FUNCTION_BLOCK FB_HeatpumpInit
VAR_IN_OUT
	MBMaster		:	ModbusRtuMasterV2_KL6x22B;
	Get				:	ST_HeatpumpGet;
END_VAR

VAR_INPUT
	ACPowerStatus	:	BOOL;
	HeatPumpID		:	BYTE;
	SFCInit			:	BOOL;
END_VAR
		
VAR
	TransmissionDone		:	BOOL;
	DataBuffer				:	ARRAY[0..50] OF WORD;
	b_MBBusy				:	BOOL;
	b_MBerr					:	BOOL;
	ui_cbRead				:	UINT;
	b_EnableTransmission	:	BOOL;
	ModbusRetryTimer		:	TON := (PT := TIME#250MS);
	ModbusStartTrigger		:	R_Trig;
	TransmissionDoneTrigger	:	F_Trig;
	MBRetryCount			:	BYTE;
	u_Counter				:	uint;
	
	SendValue		:	WORD;
	
	w_errid: Tc2_ModbusRTU.MODBUS_ERRORS;
	ResetRetryTimer: BOOL;
END_VAR
VAR_OUTPUT
END_VAR
VAR
END_VAR

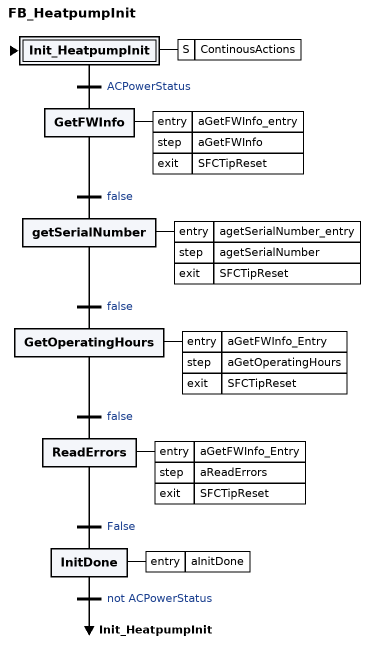
INITIAL_STEP Init_HeatpumpInit:
    ContinousActions(S);
END_STEP
TRANSITION FROM Init_HeatpumpInit TO GetFWInfo
    := ACPowerStatus;
END_TRANSITION
STEP GetFWInfo:
    aGetFWInfo_entry(P1);  // entry action
    aGetFWInfo(N);  // step action
    SFCTipReset(P0);  // exit action
END_STEP
TRANSITION FROM GetFWInfo TO getSerialNumber
    := false;
END_TRANSITION
STEP getSerialNumber:
    agetSerialNumber_entry(P1);  // entry action
    agetSerialNumber(N);  // step action
    SFCTipReset(P0);  // exit action
END_STEP
TRANSITION FROM getSerialNumber TO GetOperatingHours
    := false;
END_TRANSITION
STEP GetOperatingHours:
    aGetFWInfo_Entry(P1);  // entry action
    aGetOperatingHours(N);  // step action
    SFCTipReset(P0);  // exit action
END_STEP
TRANSITION FROM GetOperatingHours TO ReadErrors
    := false;
END_TRANSITION
STEP ReadErrors:
    aGetFWInfo_Entry(P1);  // entry action
    aReadErrors(N);  // step action
    SFCTipReset(P0);  // exit action
END_STEP
TRANSITION FROM ReadErrors TO InitDone
    := False;
END_TRANSITION
STEP InitDone:
    aInitDone(P1);  // entry action
END_STEP
TRANSITION FROM InitDone TO Init_HeatpumpInit
    := not ACPowerStatus;
END_TRANSITION

ACTION aGetFWInfo:

//ModbusStartTrigger(clk := b_EnableTransmission);

IF NOT b_enableTransmission THEN
	b_enableTransmission := TRUE;
END_IF

MBMaster.ReadRegs(	UnitID 		:= 	HeatPumpID,
					Quantity 	:= 	4,
					MBAddr		:=	1,
					cbLength 	:= 	64,
					pMemoryAddr	:=	ADR(DataBuffer),
					Execute		:=	ModbusStartTrigger.Q,
					Timeout		:=	T#250MS,		
					Busy		=>	b_MBBusy,
					Error 		=>	b_MBerr,
					cbRead 		=>	ui_cbRead,
					ErrorId		=>	w_errid
					);


TransmissionDoneTrigger(clk := b_MBBusy);

IF TransmissionDoneTrigger.q THEN
	IF NOT b_MBerr THEN
		get.HeatpumpData.i_FW_Version 		:= 	WORD_TO_INT(DataBuffer[0]);
		get.HeatpumpData.i_FW_release 		:= 	WORD_TO_INT(DataBuffer[1]);
		get.HeatpumpData.w_FW_Subrelease 	:= 	DataBuffer[2];
		get.HeatpumpData.w_FW_creationDate	:=	DataBuffer[3];
			
		TransmissionDone := TRUE;
		//done, preset for next step
		//b_EnableTransmission := FALSE;
		//ModbusStartTrigger(clk := b_EnableTransmission);
		MBRetryCount := 0;
		//ResetRetryTimer := TRUE;
		
		sfctip := TRUE;
	ELSE
		MBRetryCount := MBRetryCount + 1;
		b_EnableTransmission	:= FALSE;
		
		//if heatpump is still unreachable after 1 minute, something failed during poweron
		IF MBRetryCount > 240 THEN
			get.HeatPumpState := eHeatpumpState.ERROR;
			get.Events.b_CommError := TRUE;
		END_IF
	END_IF
END_IF



(*
IF b_EnableTransmission AND NOT b_MBBusy[0] THEN
	IF NOT b_MBerr[0] THEN
			//transmission done, process data
			get.HeatpumpData.i_FW_Version 		:= 	WORD_TO_INT(DataBuffer[0]);
			get.HeatpumpData.i_FW_release 		:= 	WORD_TO_INT(DataBuffer[1]);
			get.HeatpumpData.w_FW_Subrelease 	:= 	DataBuffer[2];
			get.HeatpumpData.w_FW_creationDate	:=	DataBuffer[3];
			
			TransmissionDone := TRUE;
			//done, preset for next step
			//b_EnableTransmission := FALSE;
			//ModbusStartTrigger(clk := b_EnableTransmission);
			MBRetryCount := 0;
	
			//sfctip := TRUE;
		ELSE
			MBRetryCount := MBRetryCount + 1;
			
			//add comm error functionality later
			IF MBRetryCount < 10 THEN
				//retry
				b_EnableTransmission	:= FALSE;
			ELSE
				//do something else
				b_EnableTransmission	:= FALSE;
			END_IF
		END_IF
	END_IF


IF TransmissionDone THEN
	sfctip := TRUE;
END_IF


IF NOT b_MBBusy[0] THEN
	IF NOT b_MBerr[0] THEN
		//transmission done, process data
		get.HeatpumpData.i_FW_Version 		:= 	WORD_TO_INT(DataBuffer[0]);
		get.HeatpumpData.i_FW_release 		:= 	WORD_TO_INT(DataBuffer[1]);
		get.HeatpumpData.w_FW_Subrelease 	:= 	DataBuffer[2];
		get.HeatpumpData.w_FW_creationDate	:=	DataBuffer[3];
		
		//done, preset for next step
		b_EnableTransmission := FALSE;
		ModbusStartTrigger(clk := b_EnableTransmission);
		MBRetryCount := 0;

		sfctip := TRUE;
	ELSE
		MBRetryCount := MBRetryCount + 1;
		
		//add comm error functionality later
		IF MBRetryCount < 10 THEN
			//retry
			b_EnableTransmission	:= FALSE;
		ELSE
			//do something else
			b_EnableTransmission	:= FALSE;
		END_IF
	END_IF
END_IF
*)
END_ACTION

ACTION aGetFWInfo_entry:
//ResetRetryTimer := TRUE;
//TransmissionDone := False;

get.HeatPumpState := eHeatpumpState.Initializing;
END_ACTION

ACTION aGetOperatingHours:


MBMaster.ReadRegs(	UnitID 		:= 	HeatPumpID,
					Quantity 	:= 	1,
					MBAddr		:=	305,
					cbLength 	:= 	1*2,
					pMemoryAddr	:=	ADR(DataBuffer),
					Execute		:=	ModbusStartTrigger.Q,
					Timeout		:=	T#250MS,		
					Busy		=>	b_MBBusy,
					Error 		=>	b_MBerr,
					cbRead 		=>	ui_cbRead,
					ErrorId		=>	w_errid
					);

TransmissionDoneTrigger(clk := b_MBBusy);

IF TransmissionDoneTrigger.q THEN
	IF NOT b_MBerr THEN
		//transmission done, process data
		
		//just use comp 1 for now. See if the others are even used
		//i think it will be a dual word value. But check later
		get.HeatpumpData.i_OperatingHours := WORD_TO_INT(DataBuffer[0]);
		
		//done, preset for next step
		b_EnableTransmission := FALSE;
//		ModbusStartTrigger(clk := b_EnableTransmission);
		MBRetryCount := 0;
		sfctip := TRUE;
	ELSE
		MBRetryCount := MBRetryCount + 1;
		b_EnableTransmission	:= FALSE;
		
		//if comm fails 5 times in a row. system is unusable
		IF MBRetryCount > 5 THEN
			get.HeatPumpState := eHeatpumpState.ERROR;
			get.Events.b_CommError := TRUE;
		END_IF
	END_IF
END_IF
END_ACTION

ACTION agetSerialNumber:



IF NOT b_enableTransmission THEN
	b_enableTransmission := TRUE;
END_IF


MBMaster.ReadRegs(	UnitID 		:= 	HeatPumpID,
					Quantity 	:= 	18,
					MBAddr		:=	80,
					cbLength 	:= 	32*2,
					pMemoryAddr	:=	ADR(DataBuffer),
					Execute		:=	ModbusStartTrigger.Q,
					Timeout		:=	T#250MS,		
					Busy		=>	b_MBBusy,
					Error 		=>	b_MBerr,
					cbRead 		=>	ui_cbRead,
					ErrorId		=>	w_errid
					);

TransmissionDoneTrigger(clk := b_MBBusy);

IF TransmissionDoneTrigger.q THEN
	IF NOT b_MBerr THEN
		FOR u_counter:=0 TO 17 BY 1 DO
			get.HeatpumpData.w_Serialnumber[u_counter]	:= 	DataBuffer[u_counter];
		END_FOR
			
		TransmissionDone := TRUE;
		//done, preset for next step
		//b_EnableTransmission := FALSE;
		//ModbusStartTrigger(clk := b_EnableTransmission);
		MBRetryCount := 0;
	
		sfctip := TRUE;
	ELSE
		MBRetryCount := MBRetryCount + 1;
		b_EnableTransmission	:= FALSE;
		
		//if comm fails 5 times in a row. system is unusable
		IF MBRetryCount > 5 THEN
			get.HeatPumpState := eHeatpumpState.ERROR;
			get.Events.b_CommError := TRUE;
		END_IF
	END_IF
END_IF

(*
IF b_EnableTransmission AND NOT b_MBBusy[2] THEN
	IF NOT b_MBerr[2] THEN
		//transmission done, process data

		
		//maybe try to put get struct directly in MBREAD pMemoryAddr later
		FOR u_counter:=0 TO 8 BY 1 DO
			get.HeatpumpData.w_Serialnumber[u_counter]	:= 	DataBuffer[u_counter];
		END_FOR
			
			TransmissionDone := TRUE;
			//done, preset for next step
			//b_EnableTransmission := FALSE;
			//ModbusStartTrigger(clk := b_EnableTransmission);
			MBRetryCount := 0;
	
			//sfctip := TRUE;
		ELSE
			MBRetryCount := MBRetryCount + 1;
			
			//add comm error functionality later
			IF MBRetryCount < 10 THEN
				//retry
				b_EnableTransmission	:= FALSE;
			ELSE
				//do something else
				b_EnableTransmission	:= FALSE;
			END_IF
		END_IF
	END_IF


IF TransmissionDone THEN
	sfctip := TRUE;
END_IF
		
				
IF NOT b_MBBusy[2] THEN
	IF NOT b_MBerr[2] THEN
		//transmission done, process data
		
		//maybe try to put get struct directly in MBREAD pMemoryAddr later
		FOR u_counter:=0 TO 8 BY 1 DO
			get.HeatpumpData.w_Serialnumber[u_counter]	:= 	DataBuffer[u_counter];
		END_FOR
		
		//done, preset for next step
		b_EnableTransmission := FALSE;
		ModbusStartTrigger(clk := b_EnableTransmission);
		MBRetryCount := 0;
		sfctip := TRUE;
	ELSE
		MBRetryCount := MBRetryCount + 1;
		
		//add comm error functionality later
		IF MBRetryCount < 10 THEN
			//retry
			b_EnableTransmission	:= FALSE;
		ELSE
			//do something else
			b_EnableTransmission	:= FALSE;
		END_IF
	END_IF
END_IF
*)
END_ACTION

ACTION agetSerialNumber_entry:
//SFCTip := FALSE;
//TransmissionDone := False;
END_ACTION

ACTION aInitDone:
SFCTip := FALSE;
IF get.HeatPumpState = eHeatPumpState.Initializing THEN
	get.HeatPumpState := eHeatPumpState.Standby;
end_if
END_ACTION

ACTION aReadErrors:
//SFCTip := FALSE;
//b_EnableTransmission	:= TRUE;
//ModbusStartTrigger(clk := b_EnableTransmission);

MBMaster.ReadRegs(	UnitID 		:= 	HeatPumpID,
					Quantity 	:= 	7,
					MBAddr		:=	950,
					cbLength 	:= 	7*2,
					pMemoryAddr	:=	ADR(DataBuffer),
					Execute		:=	ModbusStartTrigger.Q,
					Timeout		:=	T#500MS,		
					Busy		=>	b_MBBusy,
					Error 		=>	b_MBerr,
					cbRead 		=>	ui_cbRead,
					ErrorId		=>	w_errid
					);

TransmissionDoneTrigger(clk := b_MBBusy);

IF TransmissionDoneTrigger.q THEN
	IF NOT b_MBerr THEN
		//transmission done, process data
		
		ParseHeatPumpErrors(	w_Alarms1 := DataBuffer[0],
								w_Alarms2 := DataBuffer[1],
								w_Alarms3 := DataBuffer[2],
								w_Alarms4 := DataBuffer[3],
								w_Alarms5 := DataBuffer[4],
								w_Alarms6 := DataBuffer[5],
								w_Alarms7 := DataBuffer[6],
								Get := Get				
							);
		
		//done, preset for next step
		b_EnableTransmission := FALSE;
//		ModbusStartTrigger(clk := b_EnableTransmission);
		MBRetryCount := 0;
		sfctip := TRUE;
	ELSE
		MBRetryCount := MBRetryCount + 1;
		b_EnableTransmission	:= FALSE;
		
		//if comm fails 5 times in a row. system is unusable
		IF MBRetryCount > 5 THEN
			get.HeatPumpState := eHeatpumpState.ERROR;
			get.Events.b_CommError := TRUE;
		END_IF
	END_IF
END_IF
END_ACTION

ACTION ContinousActions:
//sfctip := False;
ModbusRetryTimer(in:= NOT (ModbusRetryTimer.Q OR ResetRetryTimer));
ModbusStartTrigger(clk := ModbusRetryTimer.Q);

//for initial use, get notice if 1 packet fails
IF MBRetryCount > 1 THEN
	get.Events.b_CommWarning := TRUE;
END_IF

//ResetRetryTimer := FALSE;
END_ACTION

METHOD ParseHeatPumpErrors : BOOL
VAR_INPUT
	w_Alarms1	:	WORD;
	w_Alarms2	:	WORD;
	w_Alarms3	:	WORD;
	w_Alarms4	:	WORD;
	w_Alarms5	:	WORD;
	w_Alarms6	:	WORD;
	w_Alarms7	:	WORD;
END_VAR		
VAR_IN_OUT
	get	:	ST_HeatpumpGet;	
END_VAR

get.events.b_ProbeError		:=	WORD_TO_BOOL(w_Alarms3) OR WORD_TO_BOOL(w_Alarms4) OR w_Alarms5.0;

get.events.b_PressureError		:=	w_Alarms1.0 OR	//E001: High Pressure
									w_Alarms1.1 OR //E002: Low Pressure
									w_Alarms2.3;	//E020: Inverted Pressure Transducers


get.events.b_CompressorError	:=	w_Alarms1.2 OR //E003: Compressor overheated
									w_Alarms1.7 OR //E008: Compressor underspeed
									w_Alarms1.8 OR	//E009: High disch temp
									w_Alarms1.12 OR //E013: Comp2 Overheated
									w_Alarms2.2 OR	//E019: CP2 High disch temp
									w_Alarms2.6 OR	//E023: Comp3 Overheated
									w_Alarms5.1 OR //'E801: Link Inverter1',
									w_Alarms5.2 OR //'E802: Link Inverter2',
									w_Alarms5.3 OR //'E803: Link Inverter3',
									w_Alarms5.4 OR //'E851: HWfault Inverter1',
									w_Alarms5.5 OR //'E852: HWfault Inverter2',
									w_Alarms5.6 OR //'E853: HWfault Inverter3',
									w_Alarms5.7 OR //'E861: OverCurrent Inv1',
									w_Alarms5.8 OR //'E862: OverCurrent Inv2',
									w_Alarms5.9 OR //'E863: OverCurrent Inv3',
									w_Alarms5.10 OR //'E871: High Temp Inv1',
									w_Alarms5.11 OR //'E872: High Temp Inv2',
									w_Alarms5.12 OR //'E873: High Temp Inv3',
									w_Alarms5.13 OR //'E881: Bad Voltage Inv1',
									w_Alarms5.14 OR //'E882: Bad Voltage Inv2',
									w_Alarms5.15 OR //'E883: Bad Voltage Inv3',
									w_Alarms6.0 OR //E891: Phase Seq Inv1',
									w_Alarms6.1 OR //'E892: Phase Seq Inv2',
									w_Alarms6.2 OR //'E893: Phase Seq Inv3',
									w_Alarms6.3 OR //'E901: Model err Inv1',
									w_Alarms6.4 OR //'E902: Model err Inv2',
									w_Alarms6.5 OR //'E903: Model err Inv3',
									w_Alarms6.6 OR //'E911: Ovl error Inv1',
									w_Alarms6.7 OR //'E9112: Ovl error Inv2',
									w_Alarms6.8 OR //'E913: Ovl error Inv3',
									w_Alarms6.9 OR //'E921: Overc PFC Inv1',
									w_Alarms6.10 OR //'E922: Overc PFC Inv2',
									w_Alarms6.11 OR //'E923: Overc PFC Inv3',
									w_Alarms6.12 OR //'E931: Int Com ERR Inv1',
									w_Alarms6.13 OR //'E932: Int Com ERR Inv2',
									w_Alarms6.14 OR //'E933: Int Com ERR Inv3',
									w_Alarms6.15 OR //'E941: Fault PFC Inv1',
									w_Alarms7.0 OR //E942: Fault PFC Inv2
									w_Alarms7.1 OR //'E943: Fault PFC Inv3',
									w_Alarms7.2 OR //'E951: Probe error Inv1',
									w_Alarms7.3 OR //'E952: Probe error Inv2',
									w_Alarms7.4 OR //'E953: Probe error Inv3',
									w_Alarms7.5 OR //'E961: Abnormal Cond Inv1',
									w_Alarms7.6 OR //'E962: Abnormal Cond Inv2',
									w_Alarms7.7 OR //'E963: Abnormal Cond Inv3',
									w_Alarms7.8 OR //'E971: Inv1 Eeprom Error',
									w_Alarms7.9 OR //'E972: Inv2 Eeprom Error',
									w_Alarms7.10 OR //'E973: Inv3 Eeprom Error',
									w_Alarms7.11;	//E029: CP3 High disch temp

get.events.b_ValveError		:=		w_Alarms2.11; //E041: Incongruent temps;


get.events.b_FanError			:=	w_Alarms1.2 OR //E004: Fan Overheated	
									w_Alarms1.13 OR //E014: Fan2 Overheated 
									w_Alarms2.7;	//E024: Fan3 Overheated					

get.events.b_PumpError			:=	w_Alarms1.5 OR	 	//E006: Lack of flow
									w_Alarms1.15 OR 	//E016: Pump Overheated
									w_Alarms2.9;		//E026: Pump2 Overheated

get.events.b_WaterTempError		:=	w_Alarms2.1 OR	//E018: OverTemperature
									w_Alarms1.4;	//E005: Frost

get.events.b_IOError			:=	w_Alarms2.14 OR 	//E101: IOMod1 Disconnected
									w_Alarms2.15; 		//E102: IOMod2 Disconnected
END_METHOD

ACTION SFCTipReset:
SFCTip := FALSE;
ResetRetryTimer := FALSE;
END_ACTION

END_FUNCTION_BLOCK

(* stored: Version 1.1.0.1, ProductVersion 3.1.4024.12
   POU FB_HeatpumpInit: Id {476ce5b1-079d-49a6-81a1-b35879e47147}, SpecialFunc None
   Action aGetFWInfo: Id {e9a4dfea-a599-4a4e-90dc-afedce1f3bd6}
   Action aGetFWInfo_entry: Id {383d6c30-d6b0-4e36-bada-ff8dca1c8066}
   Action aGetOperatingHours: Id {d8c00f8e-e697-4be2-97b0-ad1018da97fd}
   Action agetSerialNumber: Id {40d93614-6a67-4b9f-a168-abad2c0185a1}
   Action agetSerialNumber_entry: Id {1e1ba712-fb11-49a2-a5ce-a0fbe5851904}
   Action aInitDone: Id {12ad6ccf-5b16-42a8-98b2-b54544a101f0}
   Action aReadErrors: Id {77e18ac5-e663-45e0-b12d-1f4a75f7b609}
   Action ContinousActions: Id {e5042fe5-2127-48da-b638-5f96b5c3d27d}
   Method ParseHeatPumpErrors: Id {59c35a10-5b22-4032-94ac-2589b63a9939}
   Action SFCTipReset: Id {b429768b-902c-44a1-8eef-08ef2c1bbcc6} *)
